Yaskawa INFORM job: AAA.JBI

/JOB
//NAME AAA
//POS
///NPOS 2,0,0,0,0,0
C00000=-49329,106673,62745,4003,-50721,-4575
C00001=-46969,105372,61036,4871,-50464,-5567
//INST
///DATE 2023/02/08 11:15
///ATTR SC,RW
///GROUP1 RB1
NOP
MOVL C00000 V=10.0
MOVL C00001 V=10.0
END
